(* IEC 61131-3 sources: SIGMATEK-Jumag-Utils-Examples/typeManipulation/Class/mergeUINT, 1 file *)

(* ---- mergeUINT.st ---- *)
(*!
<Class
	Name               = "mergeUINT"
	Revision           = "0.0"
	RealtimeTask       = "false"
	CyclicTask         = "true"
	DefCyclictime      = "10 ms"
	BackgroundTask     = "false"
	Sigmatek           = "false"
	OSInterface        = "false"
	HighPriority       = "false"
	Automatic          = "false"
	UpdateMode         = "Prescan"
	SharedCommandTable = "true"
	Objectsize         = "(660,300)">
	<Channels>
	</Channels>
	<Dependencies>
		<Files>
			<File Path=".\Source\typeManipulation.c"/>
		</Files>
	</Dependencies>
	<Network Name="mergeUINT">
		<!-- List of Components in this network -->
		<Components>
			<Object
				Name       = "_base"
				Class      = "mergeBSINT"
				Position   = "(218,120)"
				Visualized = "false">
				<Channels>
					<Server Name="ClassSvr"/>
					<Server Name="LSB"/>
					<Server Name="merged"/>
					<Server Name="MSB"/>
				</Channels>
			</Object>
		</Components>
		<Comments>
		</Comments>
		<!-- List of Connections in this network -->
		<Connections>
			<Connection Source="this.ClassSvr" Destination="_base.ClassSvr" Vertices="(690,210),(518,210),"/>
			<Connection Source="this.merged" Destination="_base.merged" Vertices="(690,270),(518,270),"/>
			<Connection Source="this.MSB" Destination="_base.MSB" Vertices="(690,330),(518,330),"/>
			<Connection Source="this.LSB" Destination="_base.LSB" Vertices="(690,390),(518,390),"/>
		</Connections>
		<!-- Headerfiles -->
		<Options>
		</Options>
	</Network>
</Class>
*)
#pragma using mergeBSINT

mergeUINT : CLASS
: mergeBSINT
  //Servers:
  //Clients:
  //Variables:
		mMSB 	: UINT;
		mLSB 	: UINT;
		mMerged 	: UDINT;
  //Functions:

	FUNCTION VIRTUAL GLOBAL CyWork
		VAR_INPUT
			EAX 	: UDINT;
		END_VAR
		VAR_OUTPUT
			state (EAX) 	: UDINT;
		END_VAR;
  //Tables:
	FUNCTION @STD
		VAR_OUTPUT
			ret_code	: CONFSTATES;
		END_VAR;
	FUNCTION GLOBAL TAB @CT_;
END_CLASS;

Function Global __cdecl mergeUINT
VAR_INPUT
  MSB : UINT;
  LSB : UINT;
END_VAR
VAR_OUTPUT
  Q : UDINT;
END_VAR;

FUNCTION VIRTUAL GLOBAL mergeUINT::CyWork
	VAR_INPUT
		EAX 	: UDINT;
	END_VAR
	VAR_OUTPUT
		state (EAX) 	: UDINT;
	END_VAR

  mMSB := to_uint(MSB);
  mLSB := to_uint(LSB);

  mMerged  := mergeUINT(MSB:=mMSB, LSB:=mLSB);

  merged := to_dint(mMerged);

	state := READY;

END_FUNCTION
